// LS Electric XG5000 project: Comunica_LS
// PLC LSPLC
// module base 0 slot 1: Internal Positioning:XBF-PO02E (Open Collector Type, 2 Axis)

PROGRAM Comm (task: Scan Program)

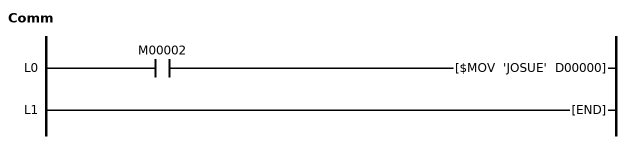
; L0
LOAD      M00002
$MOV      'JOSUE' D00000
; L1
END